FUNCTION_BLOCK LiftModel
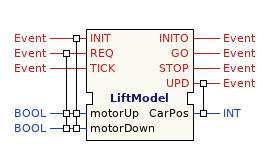
  EVENT_INPUT
    INIT WITH motorUp, motorDown;
    REQ WITH motorUp, motorDown;
    TICK;
  END_EVENT
  EVENT_OUTPUT
    INITO;
    GO;
    STOP;
    UPD WITH CarPos;
  END_EVENT
  VAR_INPUT
    motorUp : BOOL;
    motorDown : BOOL;
  END_VAR
  VAR_OUTPUT
    CarPos : INT;
  END_VAR
  VAR
    Position : DINT;
    direction : DINT;
  END_VAR
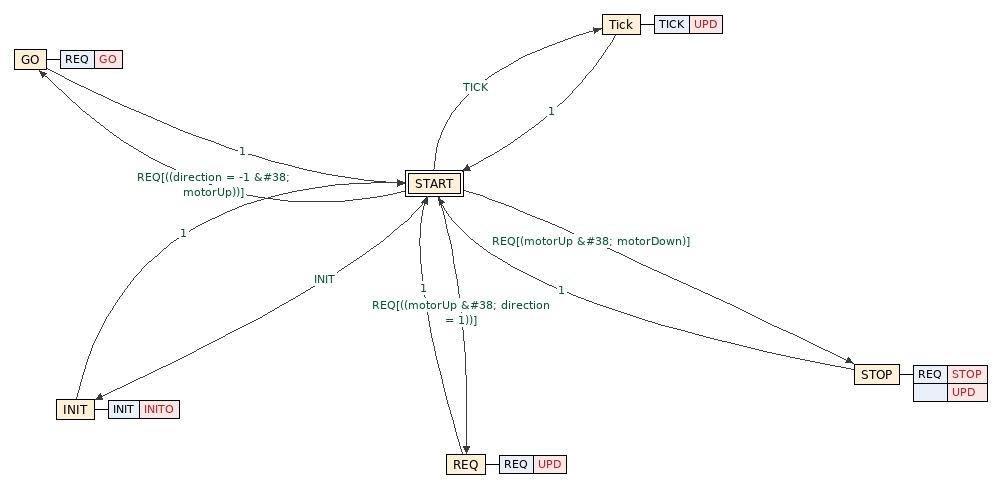
  EC_STATES
    START;
    INIT : INIT -> INITO;
    REQ : REQ -> UPD;
    Tick : TICK -> UPD;
    GO : REQ -> GO;
    STOP : REQ -> STOP, -> UPD;
  END_STATES
  EC_TRANSITIONS
    START TO INIT := INIT;
    INIT TO START := 1;
    START TO GO := REQ[((direction = -1 &#38; motorUp))];
    START TO Tick := TICK;
    Tick TO START := 1;
    START TO STOP := REQ[(motorUp &#38; motorDown)];
    GO TO START := 1;
    STOP TO START := 1;
    START TO REQ := REQ[((motorUp &#38; direction = 1))];
    REQ TO START := 1;
  END_TRANSITIONS
  ALGORITHM INIT IN ST:
Position := 1;&#38;#10;direction := 0;&#38;#10;CarPos := Position;&#38;#10;
  END_ALGORITHM
  ALGORITHM REQ IN ST:
IF motorUp THEN&#38;#10;  direction := 1;&#38;#10;ELSIF motorDown THEN&#38;#10;  direction := -1;&#38;#10;ELSE&#38;#10;  direction := 0;&#38;#10;END_IF;&#38;#10;CarPos := Position;&#38;#10;
  END_ALGORITHM
  ALGORITHM TICK IN ST:
Position := LIMIT(0, Position + direction, 6);&#38;#10;CarPos := Position;&#38;#10;
  END_ALGORITHM
END_FUNCTION_BLOCK
